TYPE ST_LoggerFactoryTags :
STRUCT
	bInformation:				BOOL;
	bWarning:					BOOL;
	bError:						BOOL;
	bPause:						BOOL;
	bHold:						BOOL;
	bComplete:					BOOL;	
END_STRUCT
END_TYPE

(* stored: Version 1.1.0.1
   DUT ST_LoggerFactoryTags: Id {39ce0b2a-9ce7-08a4-25b9-573047fbc508} *)
